(* IEC 61131-3 sources: stGeo/src, 3 files *)

(* ---- Configuration.st ---- *)
CONFIGURATION ConveyorCell
TASK Cycle (INTERVAL := T#50ms, PRIORITY := 1);
PROGRAM P1 WITH Cycle : MainProgram;
VAR_CONFIG
    P1.e_stop         AT %IX0.0 : BOOL;
    P1.running        AT %QX2.0 : BOOL;
    P1.conveyor_speed AT %QW0   : INT;
    P1.part_count     AT %MW0   : INT;
    P1.out AT %MB2 : XYPoints;
    // P1.out[0].Y AT %MW4 : INT;//Array[0..1] of INT;
END_VAR
END_CONFIGURATION

(* ---- Main.st ---- *)
PROGRAM MainProgram
VAR
    e_stop         : BOOL;   (* %IX0.0 — write TRUE to stop the line *)
    running        : BOOL;   (* %QX2.0 *)
    conveyor_speed : INT;    (* %QW0   *)
    part_count     : INT;    (* %MW0   *)
    out : XYPoints;
    Length : LREAL := 5.0;
END_VAR

out := SquarePoints();
RotateSquarePoints(Square := out);
running := NOT e_stop;
IF running THEN
    IF conveyor_speed < 100 THEN
        conveyor_speed := conveyor_speed + 5;
    ELSE
        part_count := part_count + 1;
        conveyor_speed := 0;
    END_IF;
ELSE
    conveyor_speed := 0;
END_IF;
END_PROGRAM

(* ---- Tests.st ---- *)
TEST_FUNCTION_BLOCK RotateXYTest
VAR
    Res : XYPoint;
END_VAR
    Res := RotateXY(
        X := LREAL#5.0,
        Y := LREAL#5.0,
        THETA := LREAL#90.0
    );
    ASSERT_NEAR(EXPECTED := LREAL#-5.0,
                ACTUAL := Res.X,
                DELTA := LREAL#0.015
    );
    ASSERT_NEAR(EXPECTED := LREAL#5.0,
                ACTUAL := Res.Y,
                DELTA := LREAL#0.015
    );
    Res := RotateXY(
        X := LREAL#5.0,
        Y := LREAL#5.0,
        THETA := LREAL#180.0
    );
    ASSERT_NEAR(EXPECTED := LREAL#-5.0,
                ACTUAL := Res.X,
                DELTA := LREAL#0.015
    );
    ASSERT_NEAR(EXPECTED := LREAL#-5.0,
                ACTUAL := Res.Y,
                DELTA := LREAL#0.015
    );
    Res := RotateXY(
        X := LREAL#5.0,
        Y := LREAL#5.0,
        THETA := LREAL#270.0
    );
    ASSERT_NEAR(EXPECTED := LREAL#5.0,
                ACTUAL := Res.X,
                DELTA := LREAL#0.015
    );
    ASSERT_NEAR(EXPECTED := LREAL#-5.0,
                ACTUAL := Res.Y,
                DELTA := LREAL#0.015
    );
    Res := RotateXY(
        X := LREAL#5.0,
        Y := LREAL#5.0,
        THETA := LREAL#360.0
    );
    ASSERT_NEAR(EXPECTED := LREAL#5.0,
                ACTUAL := Res.X,
                DELTA := LREAL#0.015
    );
    ASSERT_NEAR(EXPECTED := LREAL#5.0,
                ACTUAL := Res.Y,
                DELTA := LREAL#0.015
    );
END_TEST_FUNCTION_BLOCK

TEST_FUNCTION_BLOCK RotateSquarePointsTest
    VAR
       Points : XYPoints;
       Res : XYPoints;
    END_VAR
    Points := SquarePoints();
    Res := RotateSquarePoints(Square := Points);

    ASSERT_NEAR(EXPECTED := LREAL#-5.0,
                ACTUAL := Res[0].X,
                DELTA := LREAL#0.015
    );
    ASSERT_NEAR(EXPECTED := LREAL#0.0,
                ACTUAL := Res[0].Y,
                DELTA := LREAL#0.015
    );

END_TEST_FUNCTION_BLOCK

TEST_FUNCTION_BLOCK CirclesInTriangleTest
    VAR
       Expected :  ARRAY [0..65] OF XYPoint;
       Res :  ARRAY [0..65] OF XYPoint;
       Error : CirclesInTriangleError;
       I : INT;
    END_VAR
// row 0
Expected[0].X :=LREAL#0.0;
Expected[0].Y :=LREAL#0.0;
// row 1
Expected[1].X :=LREAL#- 5.0;
Expected[1].Y :=LREAL#8.660254;

Expected[2].X :=LREAL#5.0;
Expected[2].Y :=LREAL#8.660254;
// row 2
Expected[3].X :=LREAL#- 10.0;
Expected[3].Y :=LREAL#17.320508;

Expected[4].X :=LREAL#0.0;
Expected[4].Y :=LREAL#17.320508;

Expected[5].X :=LREAL#10.0;
Expected[5].Y :=LREAL#17.320508;
// row 3
Expected[6].X :=LREAL#- 15.0;
Expected[6].Y :=LREAL#25.980762;

Expected[7].X :=LREAL#- 5.0;
Expected[7].Y :=LREAL#25.980762;

Expected[8].X :=LREAL#5.0;
Expected[8].Y :=LREAL#25.980762;

Expected[9].X :=LREAL#15.0;
Expected[9].Y :=LREAL#25.980762;
// row 4
Expected[10].X :=LREAL#- 20.0;
Expected[10].Y :=LREAL#34.641016;

Expected[11].X :=LREAL#- 10.0;
Expected[11].Y :=LREAL#34.641016;

Expected[12].X :=LREAL#0.0;
Expected[12].Y :=LREAL#34.641016;

Expected[13].X :=LREAL#10.0;
Expected[13].Y :=LREAL#34.641016;

Expected[14].X :=LREAL#20.0;
Expected[14].Y :=LREAL#34.641016;
    Error := CirclesInTriangle (Points => Res);

FOR I := 0 TO 14 DO
    ASSERT_NEAR(EXPECTED := Expected[I].X,
                ACTUAL := Res[I].X,
                DELTA := LREAL#0.015
    );
END_FOR
    //Res := RotateSquarePoints(Square := Points);

    // ASSERT_NEAR(EXPECTED := LREAL#-5.0,
    //             ACTUAL := Res[0].X,
    //             DELTA := LREAL#0.015
    // );
    // ASSERT_NEAR(EXPECTED := LREAL#0.0,
    //             ACTUAL := Res[0].Y,
    //             DELTA := LREAL#0.015
    // );

END_TEST_FUNCTION_BLOCK
